// TIA Portal V17 export
// export: Created 2024-08-09T12:53:09.7986541Z, ExportSetting WithDefaults, DisplayName Totally Integrated Automation Portal, DisplayVersion V17 Update 7, DisplayName TIA Portal Openness, DisplayVersion V17 Update 7, DisplayName TIA Portal Version Control Interface, DisplayVersion V17, DisplayName STEP 7 Professional, DisplayVersion V17 Update 7, DisplayName STEP 7 Safety, DisplayVersion V17 Update 6, DisplayName WinCC Professional, DisplayVersion V17 Update 7
VAR_GLOBAL   // PLC tag table "Suiv_Lot"
END_VAR
VAR_GLOBAL CONSTANT   // user constants
   T_Nom_Tache : SInt := 20;
   T_CDCEL : SInt := 16;
   T_Num_Lot : SInt := 20;
   T_Code_Prd : SInt := 100;
   T_DESC_NET : SInt := 30;
   T_DESC_NIV : SInt := 50;
   Nbr_Max_Lots : SInt := 19;   // Nbr maximum de lots
   Nbr_Max_Tache : SInt := 59;   // Nbr maximum de taches par lot
   Niv_Tache_Max : USInt := 255;   // Niveau maximal pour une tache
   P_FinLot_Niv : USInt := 255;
   P_DebutLot_Niv : USInt := 5;
END_VAR
